TYPE TupleStruct__1:
    STRUCT
        field1: TupleStruct;
        field2: LREAL;
    END_STRUCT;
END_TYPE
